// TIA Portal V19 export
FUNCTION_BLOCK "GuardLocking"   // FB1992, F_LAD
{ S7_Optimized_Access := 'TRUE' }
// //============================================================================
// // eXcent
// //----------------------------------------------------------------------------
// // Library:
// // Tested with: V2.6
// // Engineering: TIA Portal V17
// // Restrictions: 
// // Requirements: 
// // Functionality: Interverrouillage
// //----------------------------------------------------------------------------
// // Reference to Safety Requirement Specification:
// // Safety related information: 
// //----------------------------------------------------------------------------
// // Change log table:
// // Version - Date - Signature - Expert in charge - Changes applied
// // 01 - 04.01.2021 - 0x93A71E40 - Sebastien Gros - First released version
// // 02 - 03.04.2023 - 0xAFD1BC79 - Sebastien Gros - convertion de V15-1 en V17
// // 03 - 15.08.2023 - 0x24452336 - Sebastien Gros - Ajout etat erreur de bloc
// //============================================================================
// //============================================================================
// // eXcent
// //----------------------------------------------------------------------------
// // Library:
// // Tested with: V2.6
// // Engineering: TIA Portal V17
// // Restrictions: 
// // Requirements: 
// // Functionality: GuardLocking
// //----------------------------------------------------------------------------
// // Reference to Safety Requirement Specification:
// // Safety related information: 
// //----------------------------------------------------------------------------
// // Change log table:
// // Version - Date - Signature - Expert in charge - Changes applied
// // 01 - 23.09.2024 - 0xC732AA94 - Sebastien Gros - First released version
// //============================================================================
// stored: AutoNumber false
   VAR_INPUT
      xInputSafety_1 { ExternalAccessible := 'False'; ExternalVisible := 'False'; ExternalWritable := 'False'} : Bool;   // Entree de securite 1
      xInputSafety_2 { ExternalAccessible := 'False'; ExternalVisible := 'False'; ExternalWritable := 'False'} : Bool;   // Entree de securite 2
      xStateInputSafety_1 { ExternalAccessible := 'False'; ExternalVisible := 'False'; ExternalWritable := 'False'} : Bool;   // Etat entree de securite 1
      xStateInputSafety_2 { ExternalAccessible := 'False'; ExternalVisible := 'False'; ExternalWritable := 'False'} : Bool;   // Etat entree de securite 2
      xAck { ExternalAccessible := 'False'; ExternalVisible := 'False'; ExternalWritable := 'False'} : Bool;   // Acquittement
      xAllowAck { ExternalAccessible := 'False'; ExternalVisible := 'False'; ExternalWritable := 'False'} : Bool;   // Acquittement necessaire
   END_VAR
   VAR_OUTPUT
      xStateSafety { ExternalAccessible := 'False'; ExternalVisible := 'False'; ExternalWritable := 'False'} : Bool;   // Sortie etat de securite
      stSafetyState { ExternalAccessible := 'False'; ExternalVisible := 'False'; ExternalWritable := 'False'} : "stSafetyState";   // Sortie Etat Process
   END_VAR
   VAR
      sx_Ack { ExternalAccessible := 'False'; ExternalVisible := 'False'; ExternalWritable := 'False'} : Bool;
      sx_TempAck { ExternalAccessible := 'False'; ExternalVisible := 'False'; ExternalWritable := 'False'} : Bool;
      sx_TempAckReq { ExternalAccessible := 'False'; ExternalVisible := 'False'; ExternalWritable := 'False'} : Bool;
      miDBF_Interverrouillage { ExternalAccessible := 'False'; ExternalVisible := 'False'; ExternalWritable := 'False'} : SFDOOR;
   END_VAR
   VAR CONSTANT
      cx_True : Bool := TRUE;
      cx_False : Bool := FALSE;
   END_VAR
   VAR_TEMP   // added for the SCL form of the ladder/FBD networks
      _w1 : Bool;
      _w2 : Bool;
   END_VAR
BEGIN

REGION Network 1: Validation acquitement temporaire
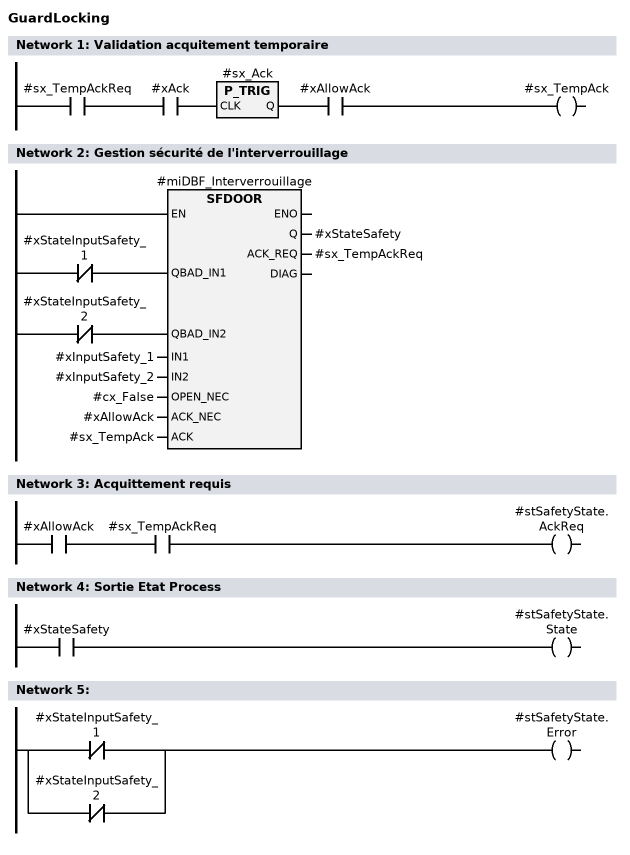
   RUNG wire#powerrail
      Contact( #sx_TempAckReq )
      Contact( #xAck )
      P_Trig( #sx_Ack )
      Contact( #xAllowAck )
      Coil( #sx_TempAck )
   END_RUNG
   // the same network as SCL:
   #_w1 := #sx_TempAckReq AND #xAck;
   #_w2 := #_w1 AND NOT #sx_Ack;   // rising edge
   #sx_Ack := #_w1;
   #sx_TempAck := #_w2 AND #xAllowAck;
END_REGION

REGION Network 2: Gestion sécurité de l'interverrouillage
   RUNG wire#powerrail
      #miDBF_Interverrouillage.SFDOOR(QBAD_IN1 := wire#w1, QBAD_IN2 := wire#w2, IN1 := #xInputSafety_1, IN2 := #xInputSafety_2, OPEN_NEC := #cx_False, ACK_NEC := #xAllowAck, ACK := #sx_TempAck, Q => #xStateSafety, ACK_REQ => #sx_TempAckReq, DIAG =>)
   END_RUNG
   RUNG wire#powerrail
      I_Contact( #xStateInputSafety_1 )
   END_RUNG wire#w1
   RUNG wire#powerrail
      I_Contact( #xStateInputSafety_2 )
   END_RUNG wire#w2
   // the same network as SCL:
   #miDBF_Interverrouillage(QBAD_IN1 := NOT #xStateInputSafety_1,   // SFDOOR
                           QBAD_IN2 := NOT #xStateInputSafety_2,
                           IN1 := #xInputSafety_1,
                           IN2 := #xInputSafety_2,
                           OPEN_NEC := #cx_False,
                           ACK_NEC := #xAllowAck,
                           ACK := #sx_TempAck,
                           Q => #xStateSafety,
                           ACK_REQ => #sx_TempAckReq);
END_REGION

REGION Network 3: Acquittement requis
   RUNG wire#powerrail
      Contact( #xAllowAck )
      Contact( #sx_TempAckReq )
      Coil( #stSafetyState.AckReq )
   END_RUNG
   // the same network as SCL:
   #stSafetyState.AckReq := #xAllowAck AND #sx_TempAckReq;
END_REGION

REGION Network 4: Sortie Etat Process
   RUNG wire#powerrail
      Contact( #xStateSafety )
      Coil( #stSafetyState.State )
   END_RUNG
   // the same network as SCL:
   #stSafetyState.State := #xStateSafety;
END_REGION

REGION Network 5
   RUNG wire#powerrail
      I_Contact( #xStateInputSafety_1 )
      wire#w1
      Coil( #stSafetyState.Error )
   END_RUNG
   RUNG wire#powerrail
      I_Contact( #xStateInputSafety_2 )
   END_RUNG wire#w1
   // the same network as SCL:
   #stSafetyState.Error := NOT #xStateInputSafety_1 OR NOT #xStateInputSafety_2;
END_REGION
END_FUNCTION_BLOCK
